{attribute 'GeneratedUsingTerminal: EL6201-0000-0017'}
{attribute addProperty BoxType "EL6201-0000-0017"}
{attribute addProperty Id "Slave_9A_DI0BOOL1Slave_9A_DI1BOOL1Slave_9A_DI2BOOL1Slave_9A_DI3BOOL1Slave_9B_DI0BOOL1Slave_9B_DI1BOOL1Slave_9B_DI2BOOL1Slave_9B_DI3BOOL1"}
{attribute addProperty CRC "4083553426"}
{attribute addProperty Size "8"}
TYPE Slave_9_Inputs_F3661492 :
STRUCT
	{attribute addProperty Name "Slave_9A_DI0"}
	Slave_9A_DI0 : BOOL;
	{attribute addProperty Name "Slave_9A_DI1"}
	Slave_9A_DI1 : BOOL;
	{attribute addProperty Name "Slave_9A_DI2"}
	Slave_9A_DI2 : BOOL;
	{attribute addProperty Name "Slave_9A_DI3"}
	Slave_9A_DI3 : BOOL;
	{attribute addProperty Name "Slave_9B_DI0"}
	Slave_9B_DI0 : BOOL;
	{attribute addProperty Name "Slave_9B_DI1"}
	Slave_9B_DI1 : BOOL;
	{attribute addProperty Name "Slave_9B_DI2"}
	Slave_9B_DI2 : BOOL;
	{attribute addProperty Name "Slave_9B_DI3"}
	Slave_9B_DI3 : BOOL;
END_STRUCT
END_TYPE

(* stored: Version 1.2.0.0, ProductVersion 3.1.4024.11
   DUT Slave_9_Inputs_F3661492: Id {ce2be45c-8b2d-495c-be36-0cc1f54f7db2} *)
